FUNCTION_BLOCK FB_StateMachine
VAR_INPUT	
	pd 							: 	REFERENCE TO ST_ProcessData;
END_VAR
VAR_OUTPUT
	iState						:	I_State := fbOffState;	
	events						:	ST_Events();
	defaultEvents 				: 	ST_Events();  			// leere Kopie
END_VAR
VAR
	fbOffState					:	FB_OffState(THIS);
	fbIdleState					:	FB_IdleState(THIS);
	fbRunningState				:	FB_RunningState(THIS);
	fbCoolDownState				:	FB_CoolDownState(THIS);
	fbErrorState				:	FB_ErrorState(THIS);
	timerTON 					: 	TON;             		// TON-Timer
	
	bStartButtonPressed    		: 	BOOL;
	bStopButtonPressed			: 	BOOL;		
	rtrigButtonSwitchOn			:	R_TRIG;
	rtrigButtonSwitchOff		:	R_TRIG;
	rtrigButtonConfirmation		:	R_TRIG;	
	strState					: 	STRING;
	
	isStartButtonEnabled		:	BOOL 	:=	TRUE;
	isStopButtonEnabled			:	BOOL 	:=	TRUE;
	timerValueToDisplay			:	INT		:= 	0;	
	bIsTimerVisible				: 	BOOL	:=  FALSE;
END_VAR

rtrigButtonSwitchOn(CLK := bStartButtonPressed);
rtrigButtonSwitchOff(CLK := bStopButtonPressed);
rtrigButtonConfirmation(CLK := pd.sensor.userConfirmation);
timerTON();

// Zuweisung von defaultEvent zu myEvent (Wertkopie)
events := defaultEvents;

generateEvents(events);

IF events.errorsDetected THEN
	iState.ErrorDetected(events.errorEvents);
END_IF 

IF events.switchOff.isTriggered THEN
	iState.UserPressedSwitchOffButton();
END_IF 

IF events.switchOn.isTriggered THEN
	iState.UserPressedSwitchOnButton();
END_IF 

IF events.confirmed.isTriggered THEN
	iState.UserPressedConfirmationButton();
END_IF 

IF events.heatIsRequested.isTriggered THEN
	iState.HeatIsRequested();
END_IF 

IF events.targetTemperatureReached.isTriggered THEN
	iState.TargetTemeperatureReached();
END_IF 

IF events.cooledDown.isTriggered THEN
	iState.WaterHasCooledDown();
END_IF

strState := iState.Name;

setButtonState();

timerTON();
timerValueToDisplay := convertTimerToDisplayValue(timerTON);

IF iState.State = E_State.IDLE AND timerTON.IN = TRUE AND timerTON.Q = FALSE THEN 	
	bIsTimerVisible := TRUE;
ELSE
	bIsTimerVisible := FALSE;
END_IF

PROPERTY INTERNAL CoolDownState : I_State
GET
CoolDownState := THIS^.fbCoolDownState;
END_GET
END_PROPERTY

PROPERTY INTERNAL ErrorState : I_State
GET
ErrorState := THIS^.fbErrorState;
END_GET
END_PROPERTY

//FB_Init ist immer implizit verfügbar und wird primär für die Initialisierung verwendet.
//Der Rückgabewert wird nicht ausgewertet. Für gezielte Einflussnahme können Sie
//die Methoden explizit deklarieren und darin mit dem Standard-Initialisierungscode 
//zusätzlichen Code bereitstellen. Sie können den Rückgabewert auswerten.
METHOD FB_Init: BOOL
VAR_INPUT    
	bInitRetains: BOOL; // TRUE: Die Retain-Variablen werden initialisiert (Reset warm / Reset kalt)    
	bInCopyCode: BOOL;  // TRUE: Die Instanz wird danach in den Kopiercode kopiert (Online-Change)
END_VAR
END_METHOD

METHOD generateEvents : BOOL
VAR_IN_OUT
	events					:	ST_Events();
END_VAR
IF (rtrigButtonSwitchOff.Q OR (rtrigButtonConfirmation.Q AND (iState.State <> E_State.OFF OR iState.State = E_State.ERROR))) THEN
	events.switchOff.isTriggered := TRUE;
ELSIF (rtrigButtonSwitchOn.Q OR (rtrigButtonConfirmation.Q AND iState.State = E_State.OFF)) THEN
	events.switchOn.isTriggered := TRUE;
ELSIF (isHeatRequested()) THEN
	events.heatIsRequested.isTriggered := TRUE;
ELSIF ((pd.sensor.temperatureFlow - pd.sensor.temperatureReturn) < GVL.configValues.temperatureDiffBacklashOff AND iState.State = E_State.COOLDOWN) THEN
	events.cooledDown.isTriggered := TRUE;
ELSIF (pd.sensor.bufferMiddleTemperature > GVL.configValues.targetTemperatureOff AND iState.State = E_State.RUNNING) THEN
	events.targetTemperatureReached.isTriggered := TRUE;
END_IF

//***** Errors *****

(* Prüfe maximalen Druck auf der Niederdruckseite über Ranco Thermostat [bar] *)
IF pd.incident.incidentLowPressure THEN
	events.errorEvents.LowPressureRefrigerationThermostat.message := CONCAT('Ranco Thermostat: zu hoher Niederdruck [bar]: ', ScaleAndRoundString(pd.sensor.pressureLow, 10));
	events.errorEvents.LowPressureRefrigerationThermostat.isTriggered := TRUE;
	events.errorsDetected := TRUE;
END_IF

(*Prüfe maximalen Druck auf der Hochdruckseite über Ranco Thermostat [bar]  *)
IF pd.incident.incidentHighPressure THEN
	events.errorEvents.HighPressureRefrigerationThermostat.message := CONCAT('Ranco Thermostat: zu hoher Hochdruck [bar]: ', ScaleAndRoundString(pd.sensor.pressureHigh, 10));
	events.errorEvents.HighPressureRefrigerationThermostat.isTriggered := TRUE;
	events.errorsDetected := TRUE;
END_IF

(* Motor-Schutzschalter hat ausgelöst *)
IF pd.incident.incidentCompressor THEN
	events.errorEvents.MotorProtectionTriggered.message := 'Motorschutzschalter hat ausgelöst';
	events.errorEvents.MotorProtectionTriggered.isTriggered := TRUE;
	events.errorsDetected := TRUE;
END_IF

(* Expansionsventil meldet Fehler *)
IF pd.incident.alarmExpansionValve THEN
	events.errorEvents.ExpansionValveTriggered.message := 'Expansionsventil meldet Fehler';
	events.errorEvents.ExpansionValveTriggered.isTriggered := TRUE;
	events.errorsDetected := TRUE;
END_IF

(* Maximaler Druckverlust des Verdampfer-Wärmetauschers [mbar] *)
IF pd.sensor.PressureDifferenceEvaporator > GVL.configValues.PressureDifferenceEvaporatorMax THEN
	events.errorEvents.PressureDiffEvaporatorTooHigh.message := CONCAT('Druckdifferenz [mbar]: ', REAL_TO_STRING(REAL_TO_INT(pd.sensor.PressureDifferenceEvaporator)));
	events.errorEvents.PressureDiffEvaporatorTooHigh.isTriggered := TRUE;
	events.errorsDetected := TRUE;
END_IF

(* Prüfe minimale Temperatur am Austritt des Verdampfer-Wärmetausschers. Triplepunkt des Wassers. [°C] *)
IF pd.sensor.TemperatureEvaporatingOut < GVL.configValues.EvaporatingTemperatureOutMin THEN
	events.errorEvents.EvaporatingTemperatureTooLow.message := CONCAT('Austritttemperatur am Verdampfer ist zu niedrig [°C]: ', ScaleAndRoundString(pd.sensor.TemperatureEvaporatingOut, 10));
	events.errorEvents.EvaporatingTemperatureTooLow.isTriggered := TRUE;
	events.errorsDetected := TRUE;
END_IF

(* Prüfe, of Wasser Durchflussmenge ausreichend ist. Mindestens 2500 Liter/Stunde *)
IF NOT pd.incident.incidentFlow THEN
	events.errorEvents.EvaporatingFlowRateTooLow.message := 'Quellwasser Durchflussmenge zu niedrig';
	events.errorEvents.EvaporatingFlowRateTooLow.isTriggered := TRUE;
	events.errorsDetected := TRUE;
END_IF

// ***** Warnings *****

(* Prüfe maximalen Druck auf der Niederdruckseite [bar] *)
IF pd.sensor.PressureLow > GVL.configValues.PressureLowMax THEN
	events.warningEvents.LowPressureRefrigerationCalc.message := CONCAT('Niederdruck: [bar]: ', ScaleAndRoundString(pd.sensor.PressureLow, 10));
	events.warningEvents.LowPressureRefrigerationCalc.isTriggered := TRUE;
ELSE
	events.warningEvents.LowPressureRefrigerationCalc.isTriggered := FALSE;
END_IF

(* Prüfe maximalen Druck auf der Hochdruckseite [bar] *)
IF pd.sensor.PressureHigh > GVL.configValues.PressureHighMax THEN
	events.warningEvents.HighPressureRefrigerationCalc.message := CONCAT('', ScaleAndRoundString(pd.sensor.PressureHigh, 10));
	events.warningEvents.HighPressureRefrigerationCalc.isTriggered := TRUE;
ELSE
	events.warningEvents.HighPressureRefrigerationCalc.isTriggered := FALSE;
END_IF

(* TANK_LEVEL_TOO_LOW *)
IF FALSE THEN
	events.warningEvents.WaterTankLevelTooLow.message := 'Wasserstand der Quelle ist zu meiedrig';
	events.warningEvents.WaterTankLevelTooLow.isTriggered := TRUE;
END_IF

(* TANK_LEVEL Data missing *)
IF FALSE THEN
	events.warningEvents.WaterTankDataMissing.message := 'Keine Daten über den Wasserstand der Quelle verfügbar';
	events.warningEvents.WaterTankDataMissing.isTriggered := TRUE;
END_IF
END_METHOD

PROPERTY INTERNAL IdleState : I_State
GET
IdleState := THIS^.fbIdleState;
END_GET
END_PROPERTY

METHOD isHeatRequested : BOOL
VAR_INPUT
END_VAR
isHeatRequested := 
	(pd.sensor.bufferTopTemperature < GVL.configValues.targetTemperatureOn) OR
	(pd.sensor.boilerHeatRequest = TRUE AND (pd.sensor.bufferTopTemperature <= pd.sensor.boilerTemperature + GVL.configValues.temperatureDiffBoilerLaden))
	AND iState.State = E_State.IDLE;
END_METHOD

METHOD isTargetTemperatureReached : BOOL
VAR_INPUT
END_VAR
// In case of State=Running the Heatpump is turned of if following condition are true
isTargetTemperatureReached := 
	pd.sensor.bufferMiddleTemperature >= GVL.configValues.targetTemperatureOff 
	AND pd.sensor.boilerHeatRequest = FALSE	
	AND iState.State = E_State.RUNNING;
END_METHOD

PROPERTY INTERNAL OffState : I_State
GET
OffState := THIS^.fbOffState;
END_GET
END_PROPERTY

PROPERTY INTERNAL RunningState : I_State
GET
RunningState := THIS^.fbRunningState;
END_GET
END_PROPERTY

METHOD setButtonState : BOOL
VAR_INPUT
END_VAR
IF iState.State <> E_State.OFF THEN 
	isStopButtonEnabled := TRUE;
	isStartButtonEnabled := FALSE;
ELSE 
	isStopButtonEnabled := FALSE;
	isStartButtonEnabled := TRUE;
END_IF

bStartButtonPressed			:= FALSE;
bStopButtonPressed			:= FALSE;
END_METHOD

METHOD INTERNAL SetState : BOOL
VAR_INPUT
	newState : I_State;
END_VAR
THIS^.iState := newState;
END_METHOD

END_FUNCTION_BLOCK

(* stored: Version 1.1.0.1
   POU FB_StateMachine: Id {c349ad72-d78c-44d0-9319-bf272785d3c6}, SpecialFunc None
   Property CoolDownState: Id {f97b0a89-973c-4c1a-a93f-bd53afa029ed}
   Get Get: Id {b6372e95-c683-40ad-a452-2ce707a937ae}
   Property ErrorState: Id {82bf1b50-5572-411a-a70d-536ddc4cc417}
   Get Get: Id {b38f7974-de10-4e45-820b-f02c66d60dde}
   Method FB_init: Id {6d3466aa-93d5-49ab-ba3a-3a7a40038459}
   Method generateEvents: Id {83685a53-198e-44e2-9f24-60ab8684b413}
   Property IdleState: Id {909b78a6-5091-4b36-9866-235bb070dd8d}
   Get Get: Id {e4d4815a-fc7b-4a73-9a7e-7c7f0b607f08}
   Method isHeatRequested: Id {5b8910d5-2963-4faa-b260-349726816464}
   Method isTargetTemperatureReached: Id {72de01e8-9221-4ced-9a58-5c631e2f44e4}
   Property OffState: Id {9baf72ca-9c89-4e21-8939-001a0e23445d}
   Get Get: Id {4045de7f-9103-414f-ae85-7d8c9bbff5c4}
   Property RunningState: Id {322a2666-716a-4153-b44f-a7d765f3afaa}
   Get Get: Id {5d6244d8-f12b-4996-a525-c240608b1a9f}
   Method setButtonState: Id {a15529d2-7ea5-42a9-a30a-580f1f9b30bd}
   Method SetState: Id {d1b82ae6-b5f8-46df-b7d5-05a5b5812d18} *)
